_CFC_ (* Continuous Function Chart, elements in execution order *)
(* 10s (5s мало) *)
(* 10s (5s мало) *)
#0 OR(SCHU_P2_2_YA1_DI6_ZKR, SCHU_P2_2_Z_NET_VH_NAPR)
#1 AND(SCHU_P2_2_SA7_DI1_A, SCHU_P2_2_AVR_A)
#2 TON_AVT:TON(IN: #1, PT: T#10s)
#3 OR(SCHU_P2_2_MP2_2_1_DI3_RUN, SCHU_P2_2_MP2_2_2_DI7_RUN)
#4 AND(#3, SCHU_P2_2_YA1_DI6_ZKR)
#5 INT_TO_TIME(ZADER_SCHU_P2_2_YA1_DI7_OTK)
#6 MUL(#5, 1000)
#7 TON_YA1_Otk:TON(IN: #4, PT: #6)
#8 AND(NOT SCHU_P2_2_MP2_2_1_DI3_RUN, NOT SCHU_P2_2_MP2_2_2_DI7_RUN)
#9 AND(#8, SCHU_P2_2_YA1_DI7_OTK)
#10 INT_TO_TIME(ZADER_SCHU_P2_2_YA1_DI6_ZKR)
#11 MUL(#10, 1000)
#12 TON_YA1_ZKR:TON(IN: #9, PT: #11)
#13 OR(SCHU_P2_2_MP2_2_1_DI3_RUN, SCHU_P2_2_MP2_2_2_DI7_RUN)
#14 AND(#13, NOT SCHU_P2_2_YA1_DI7_OTK)
#15 INT_TO_TIME(ZADER_SCHU_P2_2_YA1_DI7_OTK)
#16 MUL(#15, 1000)
#17 TON_YA1_N_OTKR:TON(IN: #14, PT: #16)
#18 AND(NOT SCHU_P2_2_MP2_2_1_DI3_RUN, NOT SCHU_P2_2_MP2_2_2_DI7_RUN)
#19 AND(#18, NOT #0)
#20 INT_TO_TIME(ZADER_SCHU_P2_2_YA1_DI6_ZKR)
#21 MUL(#20, 1000)
#22 TON_YA1_N_ZAKR:TON(IN: #19, PT: #21)
#23 OR(#7.Q, #12.Q, #17.Q, #22.Q, YA1_OTKAZ)
#24 AND(#2.Q, #23)
#25 SR_YA1_Otkaz:SR(SET1: #24, RESET: SCHU_P2_2_SB)
#26 SCHU_P2_2_Z_YA1_OTKAZ <= #25.Q1
_END_CFC_
(* the same logic as Structured Text *)
(* 10s (5s мало) *)
(* 10s (5s мало) *)
TON_AVT(IN := SCHU_P2_2_SA7_DI1_A AND SCHU_P2_2_AVR_A, PT := T#10s);
TON_YA1_Otk(IN := (SCHU_P2_2_MP2_2_1_DI3_RUN OR SCHU_P2_2_MP2_2_2_DI7_RUN) AND SCHU_P2_2_YA1_DI6_ZKR, PT := INT_TO_TIME(ZADER_SCHU_P2_2_YA1_DI7_OTK) * 1000);
TON_YA1_ZKR(IN := (NOT SCHU_P2_2_MP2_2_1_DI3_RUN AND NOT SCHU_P2_2_MP2_2_2_DI7_RUN) AND SCHU_P2_2_YA1_DI7_OTK, PT := INT_TO_TIME(ZADER_SCHU_P2_2_YA1_DI6_ZKR) * 1000);
TON_YA1_N_OTKR(IN := (SCHU_P2_2_MP2_2_1_DI3_RUN OR SCHU_P2_2_MP2_2_2_DI7_RUN) AND NOT SCHU_P2_2_YA1_DI7_OTK, PT := INT_TO_TIME(ZADER_SCHU_P2_2_YA1_DI7_OTK) * 1000);
TON_YA1_N_ZAKR(IN := (NOT SCHU_P2_2_MP2_2_1_DI3_RUN AND NOT SCHU_P2_2_MP2_2_2_DI7_RUN) AND NOT (SCHU_P2_2_YA1_DI6_ZKR OR SCHU_P2_2_Z_NET_VH_NAPR), PT := INT_TO_TIME(ZADER_SCHU_P2_2_YA1_DI6_ZKR) * 1000);
SR_YA1_Otkaz(SET1 := TON_AVT.Q AND (TON_YA1_Otk.Q OR TON_YA1_ZKR.Q OR TON_YA1_N_OTKR.Q OR TON_YA1_N_ZAKR.Q OR YA1_OTKAZ), RESET := SCHU_P2_2_SB);
SCHU_P2_2_Z_YA1_OTKAZ := SR_YA1_Otkaz.Q1;
END_PROGRAM

(* POU TZBiS/TZB/Z_YA2_Otk, CFC *)
PROGRAM Z_YA2_Otk
VAR
	SR_YA2_Otk: SR;
	TON_YA2_Rassog: TON;
	RT_Rassog: R_TRIG;
	TON_YA2_Rassog1: TON;
	TIME_DELAY: TIME;
END_VAR
VAR (* helpers for the ST form of the networks *)
	_t14 : BOOL;
	_t84 : BOOL;
	_t140 : BOOL;
END_VAR
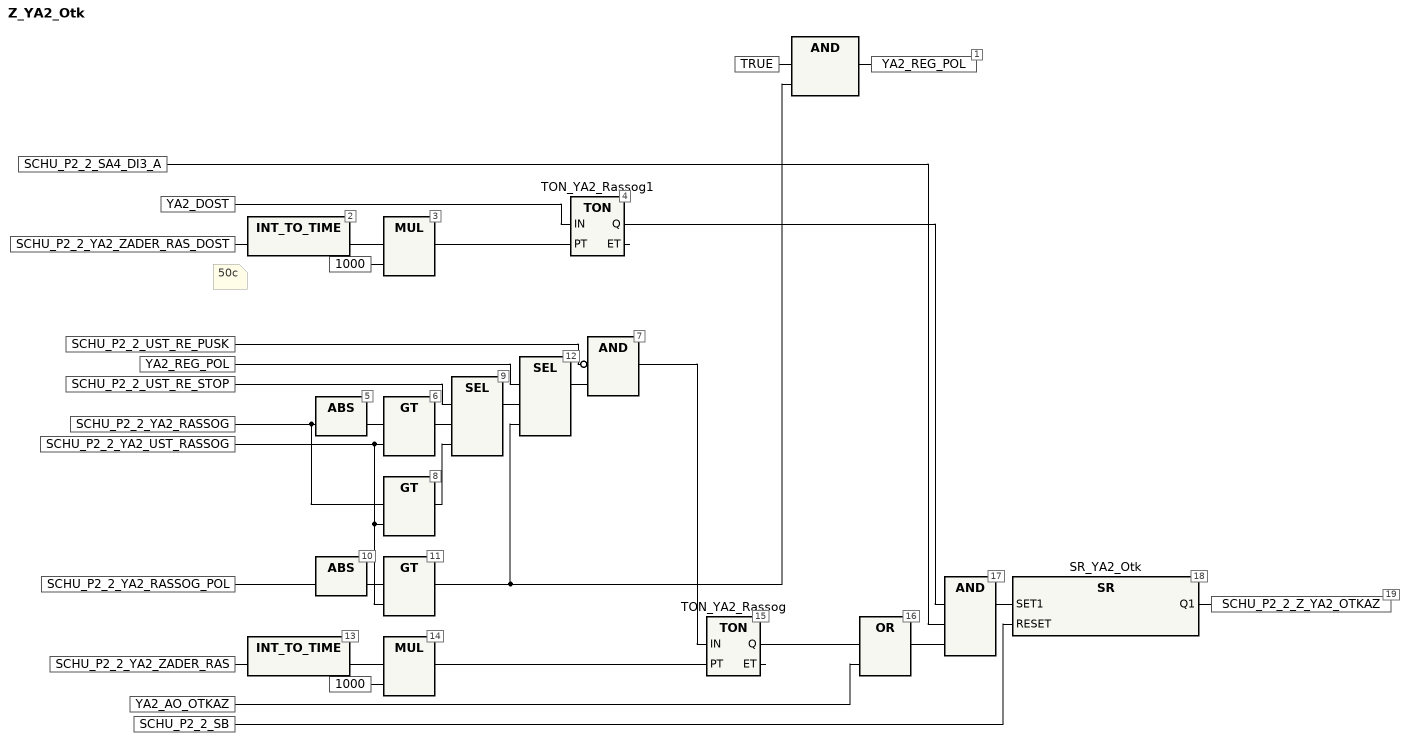
_CFC_ (* Continuous Function Chart, elements in execution order *)
(* 50с *)
#0 AND(TRUE, #11)
#1 YA2_REG_POL <= #0
#2 INT_TO_TIME(SCHU_P2_2_YA2_ZADER_RAS_DOST)
#3 MUL(#2, 1000)
#4 TON_YA2_Rassog1:TON(IN: YA2_DOST, PT: #3)
#5 ABS(SCHU_P2_2_YA2_RASSOG)
#6 GT(#5, SCHU_P2_2_YA2_UST_RASSOG)
#7 AND(NOT SCHU_P2_2_UST_RE_PUSK, #12)
#8 GT(SCHU_P2_2_YA2_RASSOG, SCHU_P2_2_YA2_UST_RASSOG)
#9 SEL(SCHU_P2_2_UST_RE_STOP, #6, #8)
#10 ABS(SCHU_P2_2_YA2_RASSOG_POL)
#11 GT(#10, SCHU_P2_2_YA2_UST_RASSOG)
#12 SEL(YA2_REG_POL, #9, #11)
#13 INT_TO_TIME(SCHU_P2_2_YA2_ZADER_RAS)
#14 MUL(#13, 1000)
#15 TON_YA2_Rassog:TON(IN: #7, PT: #14)
#16 OR(#15.Q, YA2_AO_OTKAZ)
#17 AND(#4.Q, SCHU_P2_2_SA4_DI3_A, #16)
#18 SR_YA2_Otk:SR(SET1: #17, RESET: SCHU_P2_2_SB)
#19 SCHU_P2_2_Z_YA2_OTKAZ <= #18.Q1
_END_CFC_
(* the same logic as Structured Text *)
(* 50с *)
YA2_REG_POL := TRUE AND _t14;
TON_YA2_Rassog1(IN := YA2_DOST, PT := INT_TO_TIME(SCHU_P2_2_YA2_ZADER_RAS_DOST) * 1000);
_t140 := NOT SCHU_P2_2_UST_RE_PUSK AND _t84;
_t14 := ABS(SCHU_P2_2_YA2_RASSOG_POL) > SCHU_P2_2_YA2_UST_RASSOG;
_t84 := SEL(YA2_REG_POL, SEL(SCHU_P2_2_UST_RE_STOP, ABS(SCHU_P2_2_YA2_RASSOG) > SCHU_P2_2_YA2_UST_RASSOG, SCHU_P2_2_YA2_RASSOG > SCHU_P2_2_YA2_UST_RASSOG), _t14);
TON_YA2_Rassog(IN := _t140, PT := INT_TO_TIME(SCHU_P2_2_YA2_ZADER_RAS) * 1000);
SR_YA2_Otk(SET1 := TON_YA2_Rassog1.Q AND SCHU_P2_2_SA4_DI3_A AND (TON_YA2_Rassog.Q OR YA2_AO_OTKAZ), RESET := SCHU_P2_2_SB);
SCHU_P2_2_Z_YA2_OTKAZ := SR_YA2_Otk.Q1;
END_PROGRAM

(* POU TZBiS/TZB/Z_YA3_Otk, CFC *)
PROGRAM Z_YA3_Otk
VAR
	SR_YA3_Otk: SR;
	TON_YA3_Zakl: TON;
	TON_YA3_Rassog: TON;
END_VAR
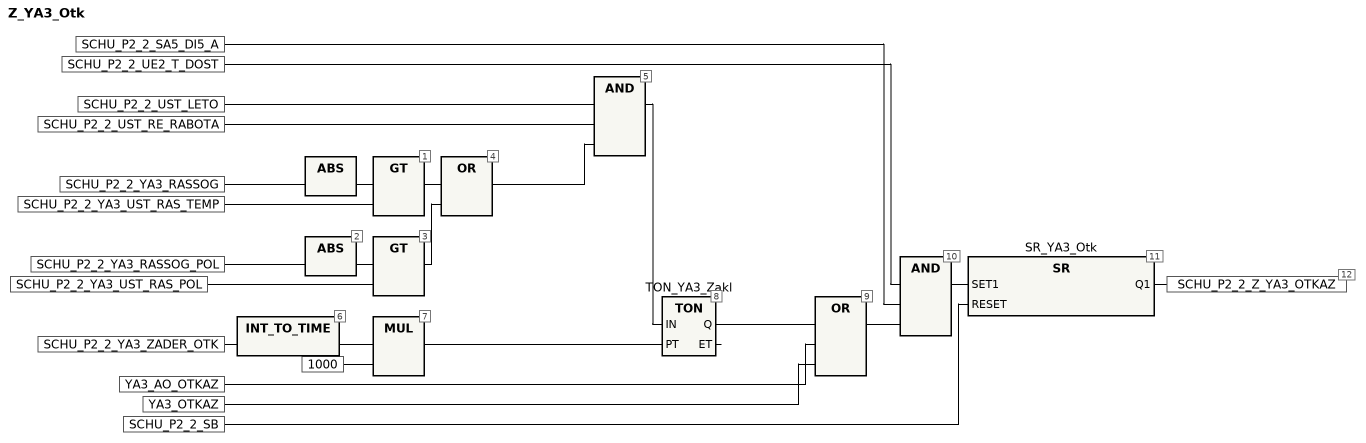
